// TIA Portal project "S7-1500 ile Zaman Kontrollü Motor Uygulaması" (V18)

(* hardware
DEVICE "S7-1500/ET200MP station_1"  S7-1500 station
   slot 0: "Rail_0"  Rack  6ES7 590-1***0-0AA0
   slot 1: "PLC_1"  CPU 1512C-1 PN  6ES7 512-1CK01-0AB0  V2.8
      slot 3: "CPU display_1"  6ES7591-1AA00-0AA0
      slot 32768: "PROFINET interface_1"  X1
         slot 32769: "Port_1"  X1 P1
         slot 32770: "Port_2"  X1 P2
      slot 34817: "Virtual CP interface port_1"  Virtual CP interface port  Virtual CP interface port
DEVICE "HMI_1"  KTP700 Basic PN
   slot 0: "HMI_1"  KTP700 Basic PN  6AV2 123-2GB03-0AX0  14.0.1.0
   slot 1: "HMI_RT_1"  KTP700 Basic PN  6AV2 123-2GB03-0AX0  14.0.1.0
   slot 5: "HMI_1.IE_CP_1"  PROFINET Interface  14.0.1.0
      slot 1: "PROFINET Interface_1"  PROFINET Interface
         slot 1: "Port_1"  Port
*)

// ===== PLC "PLC_1"  CPU 1512C-1 PN =====

VAR_GLOBAL   // PLC tag table "Default tag table"
   "Stop" AT %M0.0 : Bool;
   "Start" AT %M0.1 : Bool;
   "1. Zamanlayıcı" AT %MD100 : Time;
   "İleri" AT %Q0.0 : Bool;
   "Geri" AT %Q0.1 : Bool;
   "2. Zamanlayıcı" AT %MD200 : Time;
   "Tag_1" AT %MD120 : DInt;
   "Tag_2" AT %MD220 : DInt;
END_VAR

// folder: System blocks/Program resources

DATA_BLOCK "Zamanlayıcı_2"   // DB1
{ S7_Optimized_Access := 'TRUE' }
AUTHOR : Simatic
FAMILY : IEC
NAME : IEC_TMR
VERSION : 1.0
// stored: InstanceOfName IEC_TIMER
"IEC_TIMER"
BEGIN
END_DATA_BLOCK

DATA_BLOCK "Zamanlayıcı_1"   // DB2
{ S7_Optimized_Access := 'TRUE' }
AUTHOR : Simatic
FAMILY : IEC
NAME : IEC_TMR
VERSION : 1.0
// stored: InstanceOfName IEC_TIMER
"IEC_TIMER"
BEGIN
END_DATA_BLOCK

// folder: (top level)

ORGANIZATION_BLOCK "Main"   // OB1, LAD, ProgramCycle
TITLE = "Main Program Sweep (Cycle)"
{ S7_Optimized_Access := 'TRUE' }
VERSION : 0.1
   VAR_INPUT
      Initial_Call : Bool;   // Initial call of this OB
      Remanence : Bool;   // =True, if remanent data are available
   END_VAR
   VAR_TEMP   // added for the SCL form of the ladder/FBD networks
      _w1 : Bool;
      _w2 : Bool;
   END_VAR
BEGIN

REGION Network 1: Trafik Lambası
   // Starta basınca;
   // 20 sn ileri 30 sn geri sayacak.
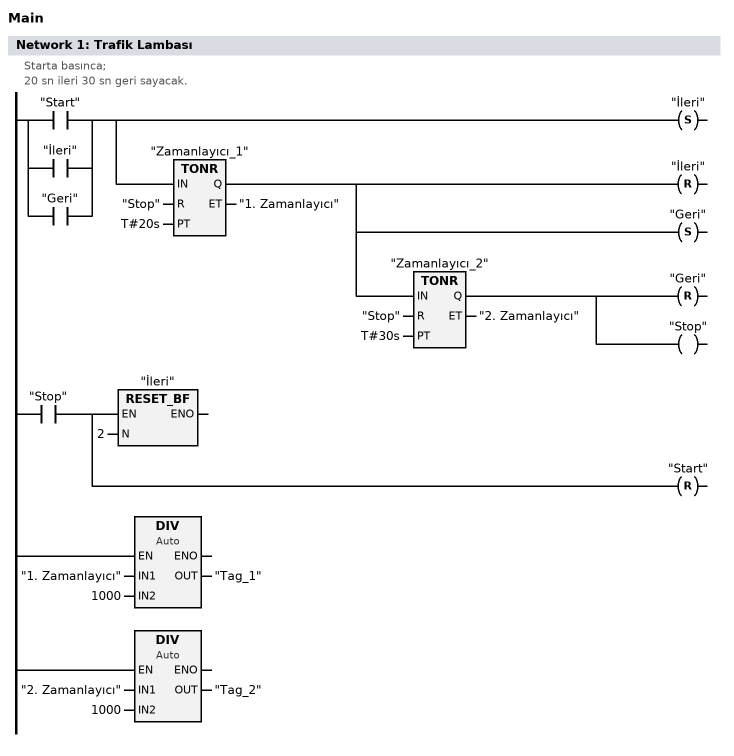
   // no SCL statement known for RBitfield: written as a call
   #_w1 := "Start" OR "İleri" OR "Geri";
   IF #_w1 THEN "İleri" := TRUE; END_IF;
   "Zamanlayıcı_1".TONR(IN := #_w1, R := "Stop", PT := T#20s, ET => "1. Zamanlayıcı");
   IF "Zamanlayıcı_1".Q THEN
       "İleri" := FALSE;
       "Geri" := TRUE;
   END_IF;
   "Zamanlayıcı_2".TONR(IN := "Zamanlayıcı_1".Q, R := "Stop", PT := T#30s, ET => "2. Zamanlayıcı");
   IF "Zamanlayıcı_2".Q THEN "Geri" := FALSE; END_IF;
   "Stop" := "Zamanlayıcı_2".Q;
   #_w2 := "Stop";
   IF #_w2 THEN
       RESET_BF(operand := "İleri", n := 2);
       "Start" := FALSE;
   END_IF;
   "Tag_1" := "1. Zamanlayıcı" / 1000;
   "Tag_2" := "2. Zamanlayıcı" / 1000;
END_REGION
END_ORGANIZATION_BLOCK

(* ===== HMI "HMI_RT_1" =====
system functions are stored by id; their names below are inferred from use
connection "Connection_1": ETHERNET, SMART_S7_1500_OMS
connection "HMI_Connection_1": ETHERNET, SMART_S7_1500_OMS

HMI tags "Default tag table"
   "Tag_ScreenNumber" : UInt, internal
   "Start_1" : Bool = PLC Start AT %M0.1, 100 ms
   "Stop" : Bool = PLC Stop AT %M0.0, 100 ms
   "2. Zamanlayıcı" : Time = PLC "2. Zamanlayıcı" AT %MD200, 100 ms
   "1. Zamanlayıcı" : Time = PLC "1. Zamanlayıcı" AT %MD100, 100 ms
   "İleri" : Bool = PLC İleri AT %Q0.0, 100 ms
   "Geri" : Bool = PLC Geri AT %Q0.1, 100 ms
   "Tag_2" : DInt = PLC Tag_2 AT %MD220, 1 s
   "Tag_1" : DInt = PLC Tag_1 AT %MD120, 1 s

graphic list "Geri Hareket": 0 'Graphic_22'; 1 'Graphic_23'

graphic list "İleri Hareket": 0 'Graphic_21'; 1 'Graphic_20'

Template "Template_1" 800x480
   Button "Exit" at 714,429 size 71x50; TextOff 'Exit'; PictureOff "ExitRuntime_KTP700_Basic_PN_TR"; PictureOn "ExitRuntime_KTP700_Basic_PN_TR"
      on Release: StopRuntime(0)
   Button "Language" at 614,429 size 71x50; TextOff 'Language'; PictureOff "ToggleLanguage_KTP700_Basic_PN_TR"; PictureOn "ToggleLanguage_KTP700_Basic_PN_TR"
      on Release: function_fb9197e8(-1)
   Button "Log on" at 514,429 size 71x50; TextOff 'Log on'; PictureOff "Login_KTP700_Basic_PN_TR"; PictureOn "Login_KTP700_Basic_PN_TR"
      on Release: function_a2a04561()
   Button "Alarms" at 114,429 size 71x50; TextOff 'Alarms'; PictureOff "AlarmDisplay_KTP700_Basic_PN_TR"; PictureOn "AlarmDisplay_KTP700_Basic_PN_TR"
      on Release: function_ef3f5d25("Alarm window_Unacknowledged", -1)
   Button "Start screen" at 14,429 size 71x50; TextOff 'Start screen'; PictureOff "NavigateHome_KTP700_Basic_PN_TR"; PictureOn "NavigateHome_KTP700_Basic_PN_TR"
      on Release: ActivateScreen("Root screen", 0)
   SymbolicIOField "Symbolic_IO_Field_Screen" at 93,9 size 600x33; TextOff '0'; TextOn '1'; TextList "TextList_ScreenNames"
      ProcessValue <- "Tag_ScreenNumber"
      on Change: ActivateScreenByNumber("Tag_ScreenNumber", 0)
   DateTimeField "HmiScreenItemData" at 695,25 size 105x25
   DateTimeField "HmiScreenItemData_1" at 695,0 size 105x25
   GraphicView "Logo" at 0,0 size 91x51; Picture "Logo of HMI_1"

screen "Root screen" 800x480, template "Template_1"
   on GenerateScreen: SetTag("Tag_ScreenNumber", 1)
   Button "Button_4" at 266,251 size 129x50; TextOff 'Start'
      on Click: InvertBit("Start_1")
      on Release: ResetBit("Start_1")
   Button "Button_1" at 266,308 size 129x50; TextOff 'Stop'
      on Press: SetBit("Stop")
      on Release: ResetBit("Stop")
   IOField "I/O field_1" at 202,188 size 129x54; FormatPattern s9999999999
      Visibility <- "Geri"
      ProcessValue <- "Tag_2"
   IOField "I/O field_2" at 202,189 size 129x54; FormatPattern s9999999999
      Visibility <- "İleri"
      ProcessValue <- "Tag_1"
   GraphicIOField "Graphic I/O field_1" at 343,188 size 96x48; PictureList "Geri Hareket"
      ProcessValue <- "Geri"
      Visibility <- "Geri"
   GraphicIOField "Graphic I/O field_2" at 343,188 size 96x48; PictureList "İleri Hareket"
      ProcessValue <- "İleri"
      Visibility <- "İleri"
*)